(* CoDeSys 2.3 export: CHECKRANGESIGNED.EXP *)

(* POU CheckRangeSigned, ST *)
FUNCTION CheckRangeSigned : DINT
VAR_INPUT
	value, lower, upper: DINT;
END_VAR
VAR
END_VAR
(* @TEXT_IMPLEMENTATION := 'ST' *)
IF value < lower THEN
	CheckRangeSigned := lower;
ELSIF value > upper THEN
	CheckRangeSigned := upper;
ELSE
	CheckRangeSigned := value;
END_IF
END_FUNCTION
